INTERFACE I_NumberResultTask EXTENDS I_Task

PROPERTY Result : LREAL
GET
END_GET
END_PROPERTY

END_INTERFACE

(* stored: Version 1.1.0.1
   Itf I_NumberResultTask: Id {d013598f-aacd-422e-9360-e2f40fdeb828}
   Property Result: Id {c980e198-8214-4e7d-83b9-984b817d2b6c}
   Get Get: Id {aaeef270-63ca-4787-8568-f31eff2ae96c} *)
